(* IEC 61131-3 sources: projects/Teichroboter/Teichroboter/butterfly/Zyklus, 7 files *)

(* ---- Kursdifferenz.st ---- *)
FUNCTION Kursdifferenz : VOID
VAR
  KOMPASS_GRAD AT %kompass_grad : INT; // Kompass Richtung, 0..3599, -1 bei Fehler @ID=7 @IN
  KURS AT %kurs_akt : INT; // aktuell gefahrener Kurs @ID=11 @IN
  KURS_DIFF AT %kurs_diff : INT; // aktuelle Kursdifferenz zum Kompass @ID=12 @IN
END_VAR
  if KOMPASS_GRAD<0 then
    // Bei Kompassfehler die Differenz auf 0 setzen
    KURS_DIFF := 0;
  else
    KURS_DIFF := KURS - KOMPASS_GRAD;
    // wenn die Differenz 180° übersteigt, dann in die andere Richtung negativ setzen
    if KURS_DIFF>1800 then
      KURS_DIFF := KURS_DIFF-3600;
    elsif KURS_DIFF<-1800 then
      KURS_DIFF := KURS_DIFF+3600;
    end_if;
  end_if;
END_FUNCTION

(* ---- Akkustand.st ---- *)
{ #define addnetworks true }
{ #define addcomments true }
{ #define addcontrolcomments false }
FUNCTION_BLOCK Akkustand
// Automatisch generiert von TeCAD, bitte Änderungen nur dort vornehmen.
{ #define title "Akkustand" }
{ #define author "TeCAD" }
VAR
  _Op0 : BYTE; // Operation 0 aktiv
  _P0 : BOOL; // Akku unter Minimum
  _P1 : BOOL; // Akku über Wiedereinschalten
END_VAR
VAR_EXTERNAL
  AKKU_NIEDRIG AT %akku_niedrig : BOOL; // Akku niedrig
  AKKU_SPANNUNG AT %akku_spannung : INT; // Spannung des Akkus
  _INIT AT %init : BOOL; // Initialisierungsvariable
END_VAR

// Initialisierung der Operationsvariablen

IF NOT _INIT THEN
  _Op0 := 2;
END_IF;
{ #define useerrortags TRUE }

// Berechnung der nicht binären Prozeßvariablen

_P0 := AKKU_SPANNUNG<1000;
_P1 := AKKU_SPANNUNG>1200;

// Ausgabe der Operationsübergänge

{ #define errortag "OP0" }
// Auswahl der Operation 0
IF _Op0 = 0 THEN
  // Übergang von Operation 0 zu Operation 1
  IF _P0 THEN
    _Op0 := 1;
  END_IF;
{ #define errortag "OP1" }
// Auswahl der Operation 1
ELSIF _Op0 = 1 THEN
  // Übergang von Operation 1 zu Operation 0
  IF (_P1 AND NOT _P0) THEN
    _Op0 := 0;
  END_IF;
{ #define errortag "INIT" }
ELSE
  // Initialisierung wenn keine Operation gesetzt ist
  _Op0 := 0;
END_IF;
{ #define useerrortags FALSE }

// Zuweisung der Operationsvariablen

// Akku niedrig
AKKU_NIEDRIG := (_Op0=1);

END_FUNCTION_BLOCK

(* ---- Antriebsfreigabe.st ---- *)
{ #define addnetworks true }
{ #define addcomments true }
{ #define addcontrolcomments false }
FUNCTION_BLOCK Antriebsfreigabe
// Automatisch generiert von TeCAD, bitte Änderungen nur dort vornehmen.
{ #define title "Antriebsfreigabe" }
{ #define author "TeCAD" }
VAR
  _Op0 : BYTE; // Operation 0 aktiv
END_VAR
VAR_EXTERNAL
  _INIT AT %init : BOOL; // Initialisierungsvariable
  ANLAGE_AUS AT %anlage_aus : BOOL; // Anlage AUS
  AKKU_NIEDRIG AT %akku_niedrig : BOOL; // Akku niedrig
  ANTRIEBSFREIGABE AT %antriebsfreigabe : BOOL; // Antriebsfreigabe erteilt
END_VAR

// Initialisierung der Operationsvariablen

IF NOT _INIT THEN
  _Op0 := 2;
END_IF;
{ #define useerrortags TRUE }

// Ausgabe der Operationsübergänge

{ #define errortag "OP0" }
// Auswahl der Operation 0
IF _Op0 = 0 THEN
  // Übergang von Operation 0 zu Operation 1
  IF (NOT ANLAGE_AUS AND NOT AKKU_NIEDRIG) THEN
    _Op0 := 1;
  END_IF;
{ #define errortag "OP1" }
// Auswahl der Operation 1
ELSIF _Op0 = 1 THEN
  // Übergang von Operation 1 zu Operation 0
  IF (ANLAGE_AUS OR AKKU_NIEDRIG) THEN
    _Op0 := 0;
  END_IF;
{ #define errortag "INIT" }
ELSE
  // Initialisierung wenn keine Operation gesetzt ist
  _Op0 := 0;
END_IF;
{ #define useerrortags FALSE }

// Zuweisung der Operationsvariablen

// Antriebsfreigabe erteilt
ANTRIEBSFREIGABE := (_Op0=1);

END_FUNCTION_BLOCK

(* ---- Kurs_fahren.st ---- *)
{ #define addnetworks true }
{ #define addcomments true }
{ #define addcontrolcomments false }
FUNCTION_BLOCK Kurs_fahren
// Automatisch generiert von TeCAD, bitte Änderungen nur dort vornehmen.
{ #define title "Kurs_fahren" }
{ #define author "TeCAD" }
VAR
  _Op0 : BYTE; // Operation 0 aktiv
  _P0 : BOOL; // Kursdifferenz positiv
  _P1 : BOOL; // Kursdifferenz negativ
  Zeit : DINT;
  _P2 : BOOL; // Rückwärtsfahrzeit abgelaufen
  _P3 : BOOL; // maximale Drehversuche abgelaufen
  _P4 : BOOL; // Kurs im Sollbereich
  _P5 : BOOL; // Störwartezeit abgelaufen
  Fahrzeit : DINT;
  _P6 : BOOL; // Fahrzeit zu lange
  Drehversuche_merk : INT;
END_VAR
VAR_EXTERNAL
  _INIT AT %init : BOOL; // Initialisierungsvariable
  ANLAGE_AUS AT %anlage_aus : BOOL; // Anlage AUS
  KURS AT %kurs_akt : INT; // aktuell gefahrener Kurs
  KOMPASS_GRAD AT %kompass_grad : INT; // Kompass Richtung, 0..3599, -1 bei Fehler
  KURS_DIFF AT %kurs_diff : INT; // aktuelle Kursdifferenz zum Kompass
  TIME_MS AT %time_ms : DINT; // Umlaufzähler in Millisekunden
  GESCHWINDIGKEIT AT %geschwindigkeit : INT; // aktuelle Sollgeschwindigkeit
  PUMPE_AUSGEKLAPPT AT %pumpe_ausgeklappt : BOOL; // Pumpe ausgeklappt
  AKKU_NIEDRIG AT %akku_niedrig : BOOL; // Akku niedrig
  STATUSTEXTNR AT %statustextnr : BYTE; // Nummer des Textes für die Anzeige am Display
  ANTRIEBSFREIGABE AT %antriebsfreigabe : BOOL; // Antriebsfreigabe erteilt
  DREHVERSUCHE AT %drehversuche : INT; // Anzahl Drehversuche als Umlaufzähler
END_VAR
VAR_TEMP
  _OV2 : BOOL;
  _OV13 : BOOL;
  _OV14 : BOOL;
  _OV5 : BOOL;
  _OV3 : BOOL;
  _OV0 : BOOL;
  _OV1 : BOOL;
  _OV4 : BOOL;
  _OV12 : BOOL;
END_VAR

// Initialisierung der Operationsvariablen

IF NOT _INIT THEN
  _Op0 := 19;
END_IF;
{ #define useerrortags TRUE }

// Berechnung der nicht binären Prozeßvariablen

_P0 := KURS_DIFF>10;
_P1 := KURS_DIFF<-10;
_P2 := (TIME_MS-Zeit)>2000;
_P3 := (DREHVERSUCHE-Drehversuche_merk)>3;
_P4 := ABS(KURS_DIFF)<150;
_P5 := (TIME_MS-Zeit)>60000;
_P6 := (TIME_MS-Fahrzeit)>120000;

// Ausgabe der Operationsübergänge

{ #define errortag "OP0" }
// Auswahl der Operation 0
IF _Op0 = 0 THEN
  // Übergang von Operation 0 zu Operation 2
  IF NOT PUMPE_AUSGEKLAPPT THEN
    _Op0 := 2;
  END_IF;
  // Übergang von Operation 0 zu Operation 1
  IF PUMPE_AUSGEKLAPPT THEN
    _Op0 := 1;
  END_IF;
{ #define errortag "OP1" }
// Auswahl der Operation 1
ELSIF _Op0 = 1 THEN
  // Übergang von Operation 1 zu Operation 15
  IF (_P2 AND PUMPE_AUSGEKLAPPT) THEN
    _Op0 := 15;
  END_IF;
  // Übergang von Operation 1 zu Operation 2
  IF (_P2 AND NOT PUMPE_AUSGEKLAPPT) THEN
    _Op0 := 2;
  END_IF;
{ #define errortag "OP2" }
// Auswahl der Operation 2
ELSIF _Op0 = 2 THEN
  // Übergang von Operation 2 zu Operation 12
  IF NOT ANTRIEBSFREIGABE THEN
    _Op0 := 12;
  END_IF;
  // Übergang von Operation 2 zu Operation 0
  IF (ANTRIEBSFREIGABE AND PUMPE_AUSGEKLAPPT) THEN
    _Op0 := 0;
  END_IF;
  // Übergang von Operation 2 zu Operation 13
  IF (ANTRIEBSFREIGABE AND NOT PUMPE_AUSGEKLAPPT AND _P6) THEN
    _Op0 := 13;
  END_IF;
  // Übergang von Operation 2 zu Operation 5
  IF (ANTRIEBSFREIGABE AND NOT PUMPE_AUSGEKLAPPT AND NOT _P6 AND _P4) THEN
    _Op0 := 5;
  END_IF;
  // Übergang von Operation 2 zu Operation 3
  IF (ANTRIEBSFREIGABE AND NOT PUMPE_AUSGEKLAPPT AND NOT _P6 AND NOT _P4 AND _P3) THEN
    _Op0 := 3;
  END_IF;
{ #define errortag "OP3" }
// Auswahl der Operation 3
ELSIF _Op0 = 3 THEN
  // Übergang von Operation 3 zu Operation 4
  IF TRUE THEN
    _Op0 := 4;
  END_IF;
{ #define errortag "OP4" }
// Auswahl der Operation 4
ELSIF _Op0 = 4 THEN
  // Übergang von Operation 4 zu Operation 12
  IF NOT ANTRIEBSFREIGABE THEN
    _Op0 := 12;
  END_IF;
  // Übergang von Operation 4 zu Operation 13
  IF (ANTRIEBSFREIGABE AND _P6) THEN
    _Op0 := 13;
  END_IF;
  // Übergang von Operation 4 zu Operation 5
  IF (ANTRIEBSFREIGABE AND NOT _P6 AND _P4) THEN
    _Op0 := 5;
  END_IF;
  // Übergang von Operation 4 zu Operation 0
  IF (ANTRIEBSFREIGABE AND NOT _P6 AND NOT _P4 AND _P3) THEN
    _Op0 := 0;
  END_IF;
{ #define errortag "OP5" }
// Auswahl der Operation 5
ELSIF _Op0 = 5 THEN
  // Übergang von Operation 5 zu Operation 12
  IF NOT ANTRIEBSFREIGABE THEN
    _Op0 := 12;
  END_IF;
  // Übergang von Operation 5 zu Operation 13
  IF (ANTRIEBSFREIGABE AND _P6) THEN
    _Op0 := 13;
  END_IF;
  // Übergang von Operation 5 zu Operation 0
  IF (ANTRIEBSFREIGABE AND NOT _P6 AND NOT _P4) THEN
    _Op0 := 0;
  END_IF;
  // Übergang von Operation 5 zu Operation 6
  IF (ANTRIEBSFREIGABE AND NOT _P6 AND _P4 AND PUMPE_AUSGEKLAPPT) THEN
    _Op0 := 6;
  END_IF;
{ #define errortag "OP6" }
// Auswahl der Operation 6
ELSIF _Op0 = 6 THEN
  // Übergang von Operation 6 zu Operation 8
  IF NOT PUMPE_AUSGEKLAPPT THEN
    _Op0 := 8;
  END_IF;
  // Übergang von Operation 6 zu Operation 7
  IF PUMPE_AUSGEKLAPPT THEN
    _Op0 := 7;
  END_IF;
{ #define errortag "OP7" }
// Auswahl der Operation 7
ELSIF _Op0 = 7 THEN
  // Übergang von Operation 7 zu Operation 17
  IF (_P2 AND PUMPE_AUSGEKLAPPT) THEN
    _Op0 := 17;
  END_IF;
  // Übergang von Operation 7 zu Operation 8
  IF (_P2 AND NOT PUMPE_AUSGEKLAPPT) THEN
    _Op0 := 8;
  END_IF;
{ #define errortag "OP8" }
// Auswahl der Operation 8
ELSIF _Op0 = 8 THEN
  // Übergang von Operation 8 zu Operation 12
  IF NOT ANTRIEBSFREIGABE THEN
    _Op0 := 12;
  END_IF;
  // Übergang von Operation 8 zu Operation 6
  IF (ANTRIEBSFREIGABE AND PUMPE_AUSGEKLAPPT) THEN
    _Op0 := 6;
  END_IF;
  // Übergang von Operation 8 zu Operation 14
  IF (ANTRIEBSFREIGABE AND NOT PUMPE_AUSGEKLAPPT AND _P6) THEN
    _Op0 := 14;
  END_IF;
  // Übergang von Operation 8 zu Operation 11
  IF (ANTRIEBSFREIGABE AND NOT PUMPE_AUSGEKLAPPT AND NOT _P6 AND _P4) THEN
    _Op0 := 11;
  END_IF;
  // Übergang von Operation 8 zu Operation 9
  IF (ANTRIEBSFREIGABE AND NOT PUMPE_AUSGEKLAPPT AND NOT _P6 AND NOT _P4 AND _P3) THEN
    _Op0 := 9;
  END_IF;
{ #define errortag "OP9" }
// Auswahl der Operation 9
ELSIF _Op0 = 9 THEN
  // Übergang von Operation 9 zu Operation 10
  IF TRUE THEN
    _Op0 := 10;
  END_IF;
{ #define errortag "OP10" }
// Auswahl der Operation 10
ELSIF _Op0 = 10 THEN
  // Übergang von Operation 10 zu Operation 12
  IF NOT ANTRIEBSFREIGABE THEN
    _Op0 := 12;
  END_IF;
  // Übergang von Operation 10 zu Operation 14
  IF (ANTRIEBSFREIGABE AND _P6) THEN
    _Op0 := 14;
  END_IF;
  // Übergang von Operation 10 zu Operation 11
  IF (ANTRIEBSFREIGABE AND NOT _P6 AND _P4) THEN
    _Op0 := 11;
  END_IF;
  // Übergang von Operation 10 zu Operation 6
  IF (ANTRIEBSFREIGABE AND NOT _P6 AND NOT _P4 AND _P3) THEN
    _Op0 := 6;
  END_IF;
{ #define errortag "OP11" }
// Auswahl der Operation 11
ELSIF _Op0 = 11 THEN
  // Übergang von Operation 11 zu Operation 12
  IF NOT ANTRIEBSFREIGABE THEN
    _Op0 := 12;
  END_IF;
  // Übergang von Operation 11 zu Operation 14
  IF (ANTRIEBSFREIGABE AND _P6) THEN
    _Op0 := 14;
  END_IF;
  // Übergang von Operation 11 zu Operation 6
  IF (ANTRIEBSFREIGABE AND NOT _P6 AND NOT _P4) THEN
    _Op0 := 6;
  END_IF;
  // Übergang von Operation 11 zu Operation 0
  IF (ANTRIEBSFREIGABE AND NOT _P6 AND _P4 AND PUMPE_AUSGEKLAPPT) THEN
    _Op0 := 0;
  END_IF;
{ #define errortag "OP12" }
// Auswahl der Operation 12
ELSIF _Op0 = 12 THEN
  // Übergang von Operation 12 zu Operation 5
  IF ANTRIEBSFREIGABE THEN
    _Op0 := 5;
  END_IF;
{ #define errortag "OP13" }
// Auswahl der Operation 13
ELSIF _Op0 = 13 THEN
  // Übergang von Operation 13 zu Operation 6
  IF TRUE THEN
    _Op0 := 6;
  END_IF;
{ #define errortag "OP14" }
// Auswahl der Operation 14
ELSIF _Op0 = 14 THEN
  // Übergang von Operation 14 zu Operation 0
  IF TRUE THEN
    _Op0 := 0;
  END_IF;
{ #define errortag "OP15" }
// Auswahl der Operation 15
ELSIF _Op0 = 15 THEN
  // Übergang von Operation 15 zu Operation 16
  IF TRUE THEN
    _Op0 := 16;
  END_IF;
{ #define errortag "OP16" }
// Auswahl der Operation 16
ELSIF _Op0 = 16 THEN
  // Übergang von Operation 16 zu Operation 0
  IF _P2 THEN
    _Op0 := 0;
  END_IF;
{ #define errortag "OP17" }
// Auswahl der Operation 17
ELSIF _Op0 = 17 THEN
  // Übergang von Operation 17 zu Operation 18
  IF TRUE THEN
    _Op0 := 18;
  END_IF;
{ #define errortag "OP18" }
// Auswahl der Operation 18
ELSIF _Op0 = 18 THEN
  // Übergang von Operation 18 zu Operation 6
  IF _P2 THEN
    _Op0 := 6;
  END_IF;
{ #define errortag "INIT" }
ELSE
  // Initialisierung wenn keine Operation gesetzt ist
  _Op0 := 12;
END_IF;
{ #define useerrortags FALSE }

// Zuweisung der Operationsvariablen

// Kurs nach vorn
_OV4 := (_Op0=8) OR (_Op0=11);
// Geschwindigkeit = vorwärts
_OV1 := (_Op0=5) OR (_Op0=11);
// Kurs nach hinten
_OV0 := (_Op0=2) OR (_Op0=5);
// Fahrzeit merken
_OV12 := (_Op0=12) OR (_Op0=13) OR (_Op0=14);
// Geschwindigkeit = rückwärts
_OV5 := (_Op0=1) OR (_Op0=4) OR (_Op0=7) OR (_Op0=10);
// Drehversuche merken
_OV14 := (_Op0=0) OR (_Op0=3) OR (_Op0=6) OR (_Op0=9);
// Geschwindigkeit=0
_OV3 := (_Op0=2) OR (_Op0=8) OR (_Op0=12) OR (_Op0=15) OR (_Op0=17);
// Kurs = Kompass
_OV13 := (_Op0=0) OR (_Op0=6) OR (_Op0=12) OR (_Op0=15) OR (_Op0=17);
// Zeit merken
_OV2 := (_Op0=5) OR (_Op0=11) OR _OV13;

// Ausgabe Sonderfunktionen und Timeraufrufe

IF _OV0 THEN
  // Kurs nach hinten
  KURS := 2800;
END_IF;
IF _OV1 THEN
  // Geschwindigkeit = vorwärts
  GESCHWINDIGKEIT := 100;
END_IF;
IF _OV2 THEN
  // Zeit merken
  Zeit := TIME_MS;
END_IF;
IF _OV3 THEN
  // Geschwindigkeit=0
  GESCHWINDIGKEIT := 0;
END_IF;
IF _OV4 THEN
  // Kurs nach vorn
  KURS := 1300;
END_IF;
IF _OV5 THEN
  // Geschwindigkeit = rückwärts
  GESCHWINDIGKEIT := -100;
END_IF;
IF (_Op0=12) THEN
  // Statustext AUS
  STATUSTEXTNR := 1;
END_IF;
IF (_Op0=0) THEN
  // Statustext DRHINT
  STATUSTEXTNR := 2;
END_IF;
IF (_Op0=5) THEN
  // Statustext FAHINT
  STATUSTEXTNR := 3;
END_IF;
IF (_Op0=6) THEN
  // Statustext DRVORN
  STATUSTEXTNR := 4;
END_IF;
IF (_Op0=11) THEN
  // Statustext FAVORN
  STATUSTEXTNR := 5;
END_IF;
IF _OV12 THEN
  // Fahrzeit merken
  Fahrzeit := TIME_MS;
END_IF;
IF _OV13 THEN
  // Kurs = Kompass
  KURS := KOMPASS_GRAD;
END_IF;
IF _OV14 THEN
  // Drehversuche merken
  Drehversuche_merk := DREHVERSUCHE;
END_IF;

END_FUNCTION_BLOCK

(* ---- Motorsteuerung.st ---- *)
{ #define addnetworks true }
{ #define addcomments true }
{ #define addcontrolcomments false }
FUNCTION_BLOCK Motorsteuerung
// Automatisch generiert von TeCAD, bitte Änderungen nur dort vornehmen.
{ #define title "Motorsteuerung" }
{ #define author "TeCAD" }
VAR
  _Op0 : BYTE; // Operation 0 aktiv
  _P0 : BOOL; // Kursdifferenz zu groß
  _P1 : BOOL; // Kursdifferenz zu klein
  Zeit : DINT;
  _P2 : BOOL; // Geschwindigkeit = 0
  _P3 : BOOL; // Drehimpuls abgelaufen
  _P4 : BOOL; // Geschwindigkeit > 0
  _P5 : BOOL; // Pausenzeit abgelaufen
  Impulsdauer : INT;
  _P6 : BOOL; // Kleiner Drehimpuls abgelaufen
END_VAR
VAR_EXTERNAL
  _INIT AT %init : BOOL; // Initialisierungsvariable
  RECHTS_PWM AT %rechts_pwm : INT; // Geschwindigkeit Motor rechts
  LINKS_PWM AT %links_pwm : INT; // Geschwindigkeit Motor links
  KURS_DIFF AT %kurs_diff : INT; // aktuelle Kursdifferenz zum Kompass
  GESCHWINDIGKEIT AT %geschwindigkeit : INT; // aktuelle Sollgeschwindigkeit
  TIME_MS AT %time_ms : DINT; // Umlaufzähler in Millisekunden
  DREHVERSUCHE AT %drehversuche : INT; // Anzahl Drehversuche als Umlaufzähler
END_VAR
VAR_TEMP
  _OV0 : BOOL;
  _OV3 : BOOL;
  _OV4 : BOOL;
  _OV9 : BOOL;
  _OV8 : BOOL;
  _OV7 : BOOL;
END_VAR

// Initialisierung der Operationsvariablen

IF NOT _INIT THEN
  _Op0 := 10;
END_IF;
{ #define useerrortags TRUE }

// Berechnung der nicht binären Prozeßvariablen

_P0 := KURS_DIFF > 150;
_P1 := KURS_DIFF < -150;
_P3 := (TIME_MS-Zeit)>Impulsdauer;
_P2 := GESCHWINDIGKEIT<0;
_P5 := (TIME_MS-Zeit)>3000;
_P4 := GESCHWINDIGKEIT>0;
_P6 := (TIME_MS-Zeit)>(Impulsdauer/5);

// Ausgabe der Operationsübergänge

{ #define errortag "OP0" }
// Auswahl der Operation 0
IF _Op0 = 0 THEN
  // Übergang von Operation 0 zu Operation 4
  IF (_P0 AND _P2) THEN
    _Op0 := 4;
  END_IF;
  // Übergang von Operation 0 zu Operation 3
  IF (_P0 AND NOT _P2) THEN
    _Op0 := 3;
  END_IF;
  // Übergang von Operation 0 zu Operation 2
  IF (NOT _P0 AND _P1 AND _P2) THEN
    _Op0 := 2;
  END_IF;
  // Übergang von Operation 0 zu Operation 1
  IF (NOT _P0 AND _P1 AND NOT _P2) THEN
    _Op0 := 1;
  END_IF;
  // Übergang von Operation 0 zu Operation 5
  IF (NOT _P0 AND NOT _P1 AND (_P2 OR _P4)) THEN
    _Op0 := 5;
  END_IF;
{ #define errortag "OP1" }
// Auswahl der Operation 1
ELSIF _Op0 = 1 THEN
  // Übergang von Operation 1 zu Operation 0
  IF NOT _P1 THEN
    _Op0 := 0;
  END_IF;
  // Übergang von Operation 1 zu Operation 6
  IF (_P1 AND _P3) THEN
    _Op0 := 6;
  END_IF;
{ #define errortag "OP2" }
// Auswahl der Operation 2
ELSIF _Op0 = 2 THEN
  // Übergang von Operation 2 zu Operation 0
  IF NOT _P1 THEN
    _Op0 := 0;
  END_IF;
  // Übergang von Operation 2 zu Operation 8
  IF (_P1 AND _P6) THEN
    _Op0 := 8;
  END_IF;
{ #define errortag "OP3" }
// Auswahl der Operation 3
ELSIF _Op0 = 3 THEN
  // Übergang von Operation 3 zu Operation 0
  IF NOT _P0 THEN
    _Op0 := 0;
  END_IF;
  // Übergang von Operation 3 zu Operation 6
  IF (_P0 AND _P3) THEN
    _Op0 := 6;
  END_IF;
{ #define errortag "OP4" }
// Auswahl der Operation 4
ELSIF _Op0 = 4 THEN
  // Übergang von Operation 4 zu Operation 0
  IF NOT _P0 THEN
    _Op0 := 0;
  END_IF;
  // Übergang von Operation 4 zu Operation 9
  IF (_P0 AND _P6) THEN
    _Op0 := 9;
  END_IF;
{ #define errortag "OP5" }
// Auswahl der Operation 5
ELSIF _Op0 = 5 THEN
  // Übergang von Operation 5 zu Operation 4
  IF (_P0 AND _P2) THEN
    _Op0 := 4;
  END_IF;
  // Übergang von Operation 5 zu Operation 3
  IF (_P0 AND NOT _P2) THEN
    _Op0 := 3;
  END_IF;
  // Übergang von Operation 5 zu Operation 2
  IF (NOT _P0 AND _P1 AND _P2) THEN
    _Op0 := 2;
  END_IF;
  // Übergang von Operation 5 zu Operation 1
  IF (NOT _P0 AND _P1 AND NOT _P2) THEN
    _Op0 := 1;
  END_IF;
  // Übergang von Operation 5 zu Operation 0
  IF (NOT _P0 AND NOT _P1 AND NOT _P2 AND NOT _P4) THEN
    _Op0 := 0;
  END_IF;
{ #define errortag "OP6" }
// Auswahl der Operation 6
ELSIF _Op0 = 6 THEN
  // Übergang von Operation 6 zu Operation 7
  IF TRUE THEN
    _Op0 := 7;
  END_IF;
{ #define errortag "OP7" }
// Auswahl der Operation 7
ELSIF _Op0 = 7 THEN
  // Übergang von Operation 7 zu Operation 0
  IF _P5 THEN
    _Op0 := 0;
  END_IF;
{ #define errortag "OP8" }
// Auswahl der Operation 8
ELSIF _Op0 = 8 THEN
  // Übergang von Operation 8 zu Operation 1
  IF TRUE THEN
    _Op0 := 1;
  END_IF;
{ #define errortag "OP9" }
// Auswahl der Operation 9
ELSIF _Op0 = 9 THEN
  // Übergang von Operation 9 zu Operation 3
  IF TRUE THEN
    _Op0 := 3;
  END_IF;
{ #define errortag "INIT" }
ELSE
  // Initialisierung wenn keine Operation gesetzt ist
  _Op0 := 0;
END_IF;
{ #define useerrortags FALSE }

// Zuweisung der Operationsvariablen

// Rechts negativ
_OV7 := (_Op0=3) OR (_Op0=4);
// Links negativ
_OV8 := (_Op0=1) OR (_Op0=2);
// Impulsdauer berechnen
_OV9 := (_Op0=0) OR (_Op0=5);
// Links aus
_OV4 := (_Op0=0) OR (_Op0=7) OR (_Op0=8);
// Rechts aus
_OV3 := (_Op0=0) OR (_Op0=7) OR (_Op0=9);
// Zeit merken
_OV0 := (_Op0=0) OR (_Op0=6) OR (_Op0=8) OR (_Op0=9);

// Ausgabe Sonderfunktionen und Timeraufrufe

IF _OV0 THEN
  // Zeit merken
  Zeit := TIME_MS;
END_IF;
IF (_Op0=1) THEN
  // Rechts positiv
  RECHTS_PWM := 100;
END_IF;
IF (_Op0=3) THEN
  // Links positiv
  LINKS_PWM := 100;
END_IF;
IF _OV3 THEN
  // Rechts aus
  RECHTS_PWM := 0;
END_IF;
IF _OV4 THEN
  // Links aus
  LINKS_PWM := 0;
END_IF;
IF (_Op0=5) THEN
  // Links Geschwindigkeit
  LINKS_PWM := GESCHWINDIGKEIT;
END_IF;
IF (_Op0=5) THEN
  // Rechts Geschwindigkeit
  RECHTS_PWM := GESCHWINDIGKEIT;
END_IF;
IF _OV7 THEN
  // Rechts negativ
  RECHTS_PWM := -120;
END_IF;
IF _OV8 THEN
  // Links negativ
  LINKS_PWM := -120;
END_IF;
IF _OV9 THEN
  // Impulsdauer berechnen
  Impulsdauer := ABS(KURS_DIFF)*5;
END_IF;
IF (_Op0=6) THEN
  // Drehversuche erhöhen
  DREHVERSUCHE := DREHVERSUCHE+1;
END_IF;

END_FUNCTION_BLOCK

(* ---- Pumpensteuerung.st ---- *)
{ #define addnetworks true }
{ #define addcomments true }
{ #define addcontrolcomments false }
FUNCTION_BLOCK Pumpensteuerung
// Automatisch generiert von TeCAD, bitte Änderungen nur dort vornehmen.
{ #define title "Pumpensteuerung" }
{ #define author "TeCAD" }
VAR
  _Op0 : BYTE; // Operation 0 aktiv
  _P0 : BOOL; // Akkuspannung zu hoch
  Zeit : DINT;
  _P1 : BOOL; // Pumpzeit vergangen
  _P2 : BOOL; // Wartezeit vergangen
  _P3 : BOOL; // Kompass im Pumpbereich
  _P4 : BOOL;
END_VAR
VAR_EXTERNAL
  _INIT AT %init : BOOL; // Initialisierungsvariable
  ANLAGE_AUS AT %anlage_aus : BOOL; // Anlage AUS
  AKKU_SPANNUNG AT %akku_spannung : INT; // Spannung des Akkus
  TIME_MS AT %time_ms : DINT; // Umlaufzähler in Millisekunden
  PUMPE_EIN AT %pumpe_ein : BOOL; // Pumpe einschalten
  AKKU_NIEDRIG AT %akku_niedrig : BOOL; // Akku niedrig
  KURS AT %kurs_akt : INT; // aktuell gefahrener Kurs
  PUMPE_AUSGEKLAPPT AT %pumpe_ausgeklappt : BOOL; // Pumpe ausgeklappt
  KOMPASS_GRAD AT %kompass_grad : INT; // Kompass Richtung, 0..3599, -1 bei Fehler
END_VAR
VAR_TEMP
  _OV0 : BOOL;
END_VAR

// Initialisierung der Operationsvariablen

IF NOT _INIT THEN
  _Op0 := 4;
END_IF;
{ #define useerrortags TRUE }

// Berechnung der nicht binären Prozeßvariablen

_P0 := AKKU_SPANNUNG>1420;
_P1 := (TIME_MS-Zeit)>3000;
_P2 := (TIME_MS-Zeit)>20000;
_P3 := KOMPASS_GRAD<1800 AND KOMPASS_GRAD>700;

// Ausgabe der Operationsübergänge

{ #define errortag "OP0" }
// Auswahl der Operation 0
IF _Op0 = 0 THEN
  // Übergang von Operation 0 zu Operation 1
  IF (_P0 OR (NOT AKKU_NIEDRIG AND NOT ANLAGE_AUS AND NOT PUMPE_AUSGEKLAPPT AND _P3)) THEN
    _Op0 := 1;
  END_IF;
{ #define errortag "OP1" }
// Auswahl der Operation 1
ELSIF _Op0 = 1 THEN
  // Übergang von Operation 1 zu Operation 0
  IF (AKKU_NIEDRIG OR ANLAGE_AUS) THEN
    _Op0 := 0;
  END_IF;
  // Übergang von Operation 1 zu Operation 2
  IF (NOT AKKU_NIEDRIG AND NOT ANLAGE_AUS AND _P1) THEN
    _Op0 := 2;
  END_IF;
{ #define errortag "OP2" }
// Auswahl der Operation 2
ELSIF _Op0 = 2 THEN
  // Übergang von Operation 2 zu Operation 3
  IF TRUE THEN
    _Op0 := 3;
  END_IF;
{ #define errortag "OP3" }
// Auswahl der Operation 3
ELSIF _Op0 = 3 THEN
  // Übergang von Operation 3 zu Operation 0
  IF _P2 THEN
    _Op0 := 0;
  END_IF;
{ #define errortag "INIT" }
ELSE
  // Initialisierung wenn keine Operation gesetzt ist
  _Op0 := 0;
END_IF;
{ #define useerrortags FALSE }

// Zuweisung der Operationsvariablen

// Pumpe einschalten
PUMPE_EIN := (_Op0=1);
// Zeit merken
_OV0 := (_Op0=0) OR (_Op0=2);

// Ausgabe Sonderfunktionen und Timeraufrufe

IF _OV0 THEN
  // Zeit merken
  Zeit := TIME_MS;
END_IF;

END_FUNCTION_BLOCK

(* ---- Zyklus.st ---- *)
{ #use "Akkustand.st" }
{ #use "Antriebsfreigabe.st" }
{ #use "Kurs_fahren.st" }
{ #use "Kursdifferenz.st" }
{ #use "Motorsteuerung.st" }
{ #use "Pumpensteuerung.st" }
FUNCTION_BLOCK Zyklus
// automatisch generiert von TERANiS-Studio, bitte Änderungen nur dort vornehmen.
{ #define title "Zyklus" }
{ #define author "TERANiS" }
VAR
  I_Akkustand : Akkustand;
  I_Antriebsfreigabe : Antriebsfreigabe;
  I_Kurs_fahren : Kurs_fahren;
  I_Motorsteuerung : Motorsteuerung;
  I_Pumpensteuerung : Pumpensteuerung;
  _INIT AT %init : BOOL;
END_VAR
  I_Akkustand(); // Akkustand.prp
  I_Antriebsfreigabe(); // Antriebsfreigabe.prp
  I_Kurs_fahren(); // Kurs_fahren.prp
  Kursdifferenz(); // Kursdifferenz.st
  I_Motorsteuerung(); // Motorsteuerung.prp
  I_Pumpensteuerung(); // Pumpensteuerung.prp
  // Initialisierungsvariable setzen
  _INIT := TRUE;
END_FUNCTION_BLOCK
